// TIA Portal V20 export
TYPE "LER_typeStep"
// stored: Access Published
   STRUCT
      action1 { ExternalAccessible := 'False'; ExternalVisible := 'False'; ExternalWritable := 'False'} : Array[0..9999] of Bool;
      action2 : Array[0..9999] of Bool;
      action3 : Array[0..9999] of Bool;
      action4 : Array[0..9999] of Bool;
      transition1 { ExternalAccessible := 'False'; ExternalVisible := 'False'; ExternalWritable := 'False'} : Array[0..9999] of Bool;
      transition2 : Array[0..9999] of Bool;
      transition3 : Array[0..9999] of Bool;
      transition4 : Array[0..9999] of Bool;
   END_STRUCT;
END_TYPE
